(* CODESYS project fill.project

Project tree, tasks and I/O mapping:
  Device : 750-8111 PFC100, WAGO, order no. 750-8111, version 6.2.0.1
    application Application
      libraries: Standard, 3.5.18.0 (System)
      task DefaultTask (cyclic, interval T#10ms, priority 8) calls PLC_PRG
      Data types/
      Global Variables/
        global variables Variablen_Konfiguration
        global variables Globale_Variablen
      POUs/
        function block VALVE_VALID [CFC]
        function block BEMPTY [CFC]
        function block calc_progress [ST]
        function block calibrate [ST]
        function block ClearCommands [ST]
        function block conv_levelsensor [ST]
        function block copy_temperature [ST]
        function block EMPTY [CFC]
        function block FILL [CFC]
        function block FLUSH [CFC]
        function block WATERWARNING [CFC]
        program PLC_PRG [CFC]
        function block run_command [ST]
        function block SELECT_VALVE [ST]
        function block smooth [ST]
        function block TIMEOUT [ST]
        function block TIMEOUT_FB [CFC]
        Configuration/
          program MODBUS_CONFIGURATION [ST]
      Visualizations/
        visualisation temp
        visualisation PLC_VISU
      trace Sampling_Trace (task ): 
    Kbus : Kbus, WAGO, version 2.1.0.1
        unmapped channels: K-BUS diagnostics
      _750_497_16 : 750-497#16, WAGO, order no. 750-497, version 2.0.0.9
          unmapped channels: _PW 1, _PW 2, _PW 3, _PW 4, _PW 5, _PW 6, _PW 7, _PW 8
      _750_460_08 : 750-460#08, WAGO, order no. 750-460, version 2.0.0.9
          unmapped channels: _IINT 1, _IINT 2, _IINT 3, _IINT 4
      _750_430 : 750-430, WAGO, order no. 750-430, version 2.0.0.14
          unmapped channels: _IN
      _750_1504_1 : 750-1504, WAGO, order no. 750-1504, version 2.0.0.14
          unmapped channels: _OUT
      _750_1504 : 750-1504, WAGO, order no. 750-1504, version 2.0.0.14
          unmapped channels: _OUT
  GlobalImagePool
  text list GlobalTextList
*)

// Device/Application/Global Variables/Variablen_Konfiguration
VAR_CONFIG
END_VAR

// Device/Application/Global Variables/Globale_Variablen
VAR_GLOBAL

	(* 8x AI 0-10V *)
	ACTWEIGHT 		AT %IW0:INT; (* 0 Actual reservoir weight in digital units, evtl. with status byte *)
	RAINFILL1 		AT %IW1:INT; (* 1 Rainbucket filling in digital units, 2.2V / 0.305mV/DU is 100% *)
	RAINFILL2 		AT %IW2:INT; (* 2 Rainbucket filling in digital units, 2.2V / 0.305mV/DU is 100% *)
	AUX0				AT %IW3:INT;
	AUX1				AT %IW4:INT;
	AUX2				AT %IW5:INT;
	AUX3				AT %IW6:INT;
	AUX4				AT %IW7:INT;

	(*4x Pt100 *)
	PT100_1			AT %IW8:INT;
	PT100_2			AT %IW9:INT;
	PT100_3			AT %IW10:INT;
	PT100_4			AT %IW11:INT;

	(* 8x DI *)
	BTN_RESET_HW	AT %IX12.0:BOOL; (* 1 Stops the current action and cancels Warnings*)
	BTN_EMPTY_HW	AT %IX12.1:BOOL; (* 2 Empties the reservoir *)
	WATERWARN1	AT %IX12.4:BOOL; (* 5 Water sensor under mounting wall (not implemented) *)
	WATERWARN2	AT %IX12.5:BOOL; (* 6 Water sensor in fridge (not implemented) *)


	(* 8x DO *)
	P1_FWD 			AT %QX0.0:BOOL; (* Main pump forward *)
	P1_BCK 			AT %QX0.1:BOOL; (* Main pump backward *)
	VRin 				AT %QX0.2:BOOL; (* Flush / Fill selector valve VRin *)
	VRout 				AT %QX0.3:BOOL; (* 2/2 Valve at reservoir outlet, connected with pump 2 *)
	VRfridge 			AT %QX0.4:BOOL; (* 3/2 valve Fridge / Valve *)
	YSI600R_PWR	AT %QX0.5:BOOL; (* Relais to power YSI600R *)
	(*AUX_DO1  		AT %QX1.7:BOOL; *)

	(* 8x DO *)
	WWARN_LED		AT %QX1.0:BOOL;
	TIMEOUT_LED 	AT %QX1.1:BOOL; (* Indicates an unwanted timeout at empty or fill*)
	RUNNING_LED 	AT %QX1.2:BOOL; (* Indicates an unwanted timeout at empty or fill*)


	(* 8x DO - Input Valves, defined in SELECT_VALVE
		%QX1.0..7
	*)
	(* 8x DO - Input Valves, defined in SELECT_VALVE
		%QX1.8..15
	*)


	(* MERKER *)
	(* Commands *)
	BTN_RESET		AT %MX0.0:BOOL; (* Resets the current action *)
	BTN_FLUSH		AT %MX0.1:BOOL; (* Starts the fill sequence, when valve is selected*)
	BTN_FILL 			AT %MX0.2:BOOL; (* Starts the fill sequence when ACTWEIGHT<TGTWEIGHT*)
	BTN_EMPTY		AT %MX0.3:BOOL; (* Starts the empty sequence when ACTWEIGHT>TGTWEIGHT*)
       BTN_FRIDGE		AT %MX0.4:BOOL; (* Sets the fridge, use together with BTN_EMPTY*)
	BTN_BEMPTY		AT %MX0.5:BOOL; (* Runs backward empty (not implemented yet*)
	BTN_YSI600R		AT %MX0.6:BOOL; (* Switches the YSI600R on during flush*)
	BTN_CALIB		AT %MX0.7:BOOL; (* Calibrates the scale *)
	BTN_RAISE_TIMEOUT AT %MX0.8:BOOL; (* Indicates that a timeout should be raised *)
	(* Command arguments *)
	VALVE 				AT %MW1:INT; (*The actual valve number*)
	TGTWEIGHT 		AT %MW2:REAL;  (*target weight in ml *)
	TIMEOUT_VAL 	AT %MW4:TIME := t#10s; (* The timeout value *)

	(* Status *)
	ST_RUNNING		AT %MX6.0:BOOL;
	ST_TIMEOUT		AT %MX6.1:BOOL;
	ST_WWARN		AT %MX6.2:BOOL;
	ST_READY		AT %MX6.3:BOOL;
	ST_RESET		AT %MX6.4:BOOL;

	PROGRESS		AT %MW7:INT;
	AVGWEIGHT		AT %MW8:REAL := -1E10; (* Average weight in ml *)
	ELAPSED 			AT %MW10:TIME; (* The elapsed time *)
	RAINFILL1_out	AT %MW12:REAL;
	RAINFILL2_out	AT %MW14:REAL;
	(*Settings*)
	MAX_VALVE		AT %MW16:INT := 12; (* Maximum number of available valves *)
	WSMOOTH		AT %MW17:INT := 10; (* Smooth factor for low pass filter *)
	CALIB_OFFSET	AT %MW18:REAL := 0; (* Offset in digital units, when empty *)
	CALIB_GAIN		AT %MW20:REAL := 0.153; (* Gain of weight calibration in ml/DU *)

	(* Temperature *)
	TEMP1			     AT %MW22:INT;
	TEMP2			     AT %MW23:INT;
       TEMP3                  AT %MW24:INT;
       TEMP4                  AT %MW25:INT;

	START_WEIGHT: REAL;

END_VAR

// Device/Application/POUs/PLC_PRG
PROGRAM PLC_PRG
VAR

	VALVE_SELECTOR: SELECT_VALVE;
	WATERWARNING: WATERWARNING;
	weight_smooth: smooth;
	conv_rf1: conv_levelsensor;
	conv_rf2: conv_levelsensor;
	START_WEIGHT: REAL;
	CMD: run_command;
	_timeout: TIMEOUT;
	CP_TEMP: copy_temperature;
END_VAR
VAR // added by the converter: edge detectors and wires of the graphical bodies
    _w1 : ANY;
END_VAR

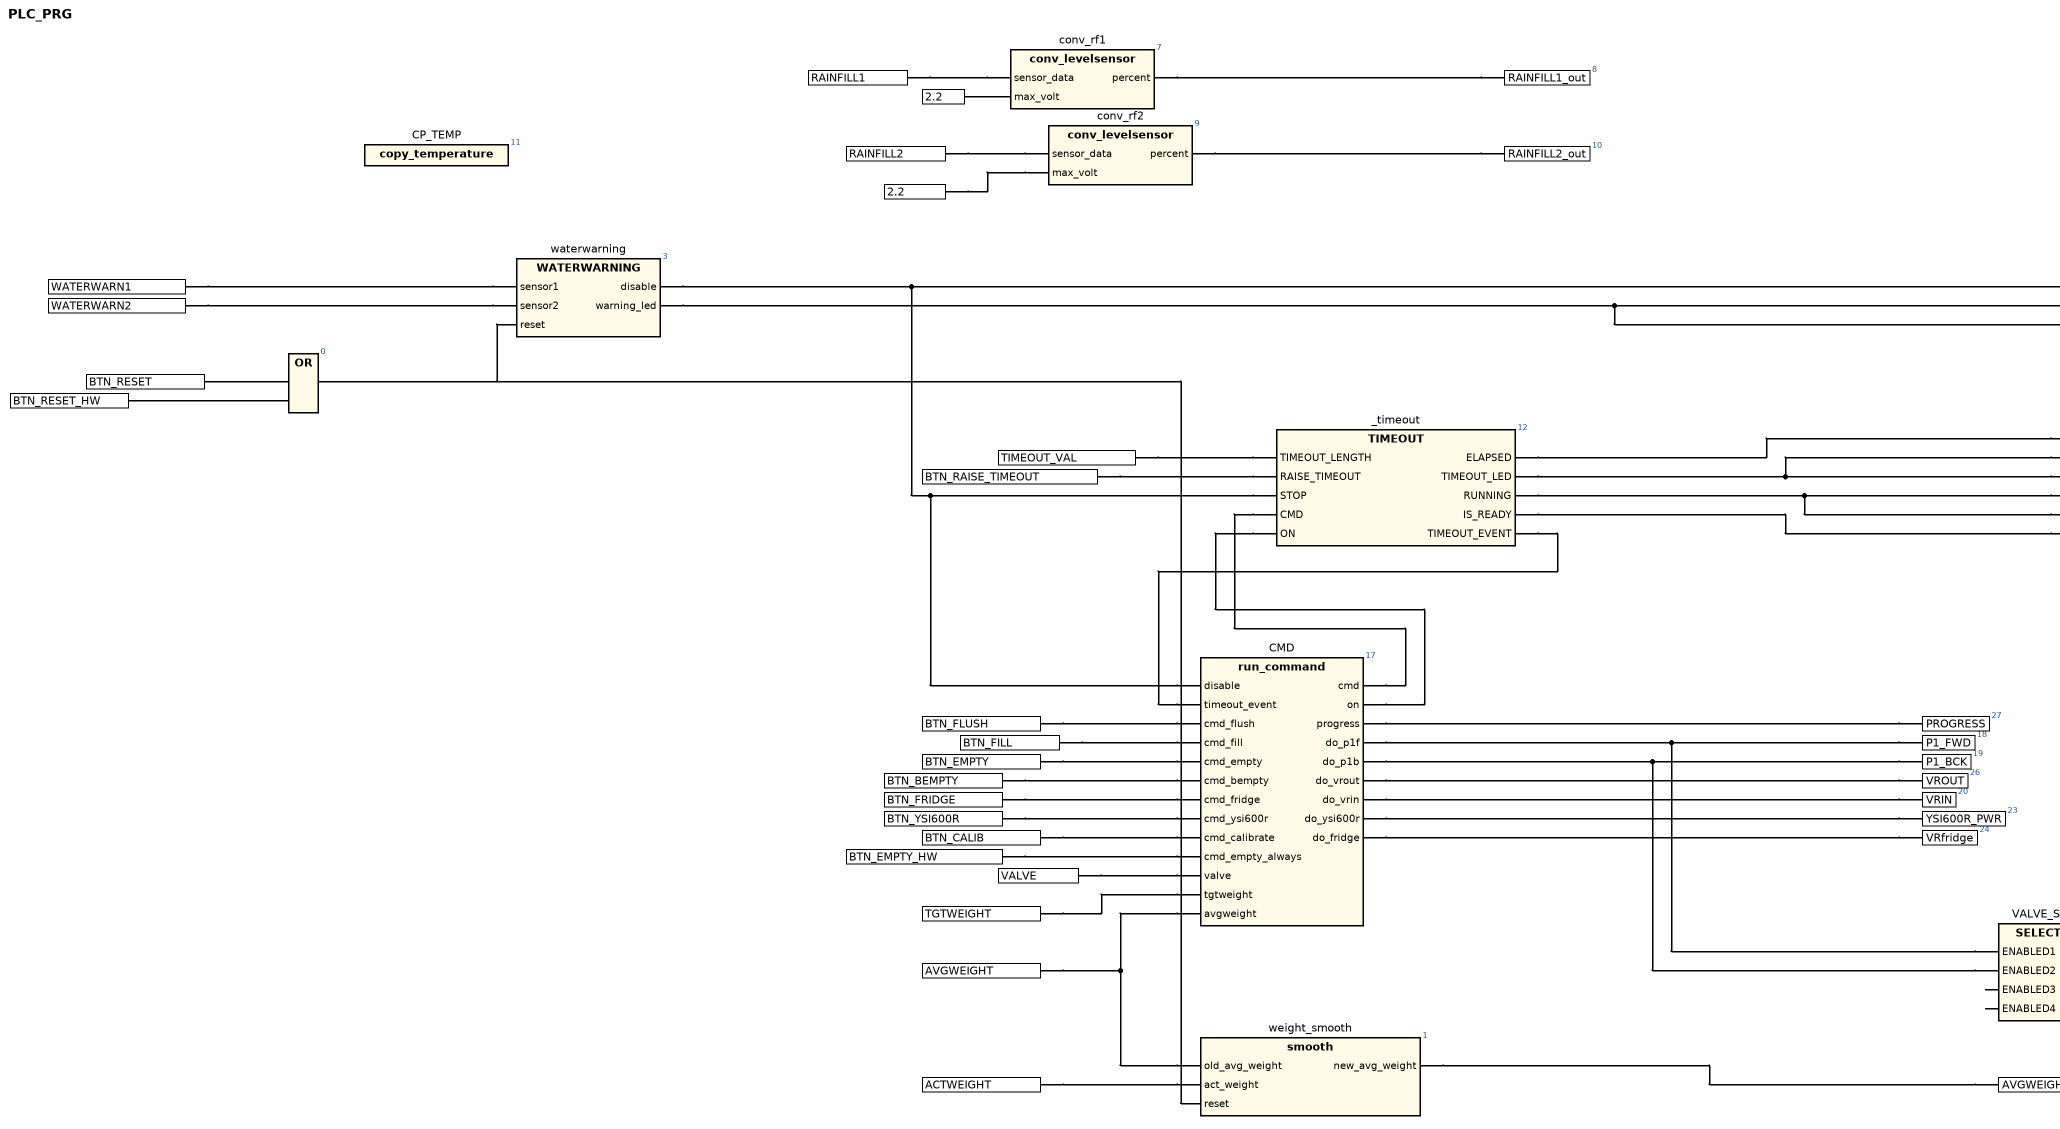
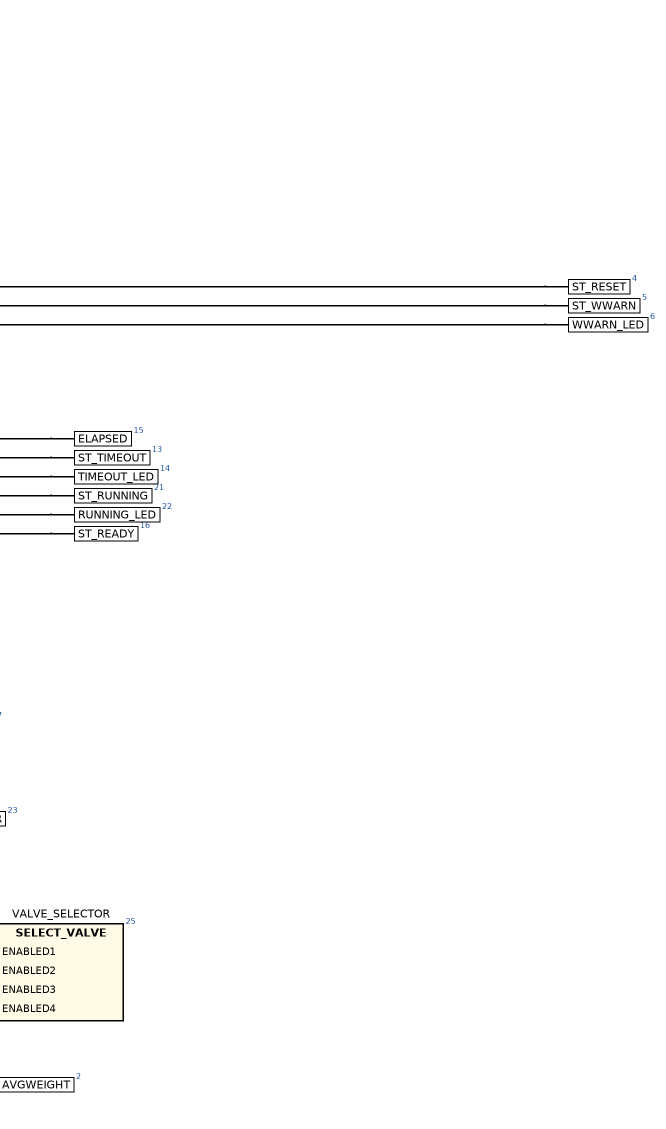
_w1 := BTN_RESET OR BTN_RESET_HW;
weight_smooth(old_avg_weight := AVGWEIGHT, act_weight := ACTWEIGHT, reset := _w1); // smooth
AVGWEIGHT := weight_smooth.new_avg_weight;
waterwarning(sensor1 := WATERWARN1, sensor2 := WATERWARN2, reset := _w1);
ST_RESET := waterwarning.disable;
ST_WWARN := waterwarning.warning_led;
WWARN_LED := waterwarning.warning_led;
conv_rf1(sensor_data := RAINFILL1, max_volt := 2.2); // conv_levelsensor
RAINFILL1_out := conv_rf1.percent;
conv_rf2(sensor_data := RAINFILL2, max_volt := 2.2); // conv_levelsensor
RAINFILL2_out := conv_rf2.percent;
CP_TEMP(); // copy_temperature
_timeout(
    TIMEOUT_LENGTH := TIMEOUT_VAL,
    RAISE_TIMEOUT := BTN_RAISE_TIMEOUT,
    STOP := waterwarning.disable,
    CMD := CMD.cmd,
    ON := CMD.on); // TIMEOUT
ST_TIMEOUT := _timeout.TIMEOUT_LED;
TIMEOUT_LED := _timeout.TIMEOUT_LED;
ELAPSED := _timeout.ELAPSED;
ST_READY := _timeout.IS_READY;
CMD(
    disable := waterwarning.disable,
    timeout_event := _timeout.TIMEOUT_EVENT,
    cmd_flush := BTN_FLUSH,
    cmd_fill := BTN_FILL,
    cmd_empty := BTN_EMPTY,
    cmd_bempty := BTN_BEMPTY,
    cmd_fridge := BTN_FRIDGE,
    cmd_ysi600r := BTN_YSI600R,
    cmd_calibrate := BTN_CALIB,
    cmd_empty_always := BTN_EMPTY_HW,
    valve := VALVE,
    tgtweight := TGTWEIGHT,
    avgweight := AVGWEIGHT); // run_command
P1_FWD := CMD.do_p1f;
P1_BCK := CMD.do_p1b;
VRIN := CMD.do_vrin;
ST_RUNNING := _timeout.RUNNING;
RUNNING_LED := _timeout.RUNNING;
YSI600R_PWR := CMD.do_ysi600r;
VRfridge := CMD.do_fridge;
VALVE_SELECTOR(ENABLED1 := CMD.do_p1f, ENABLED2 := CMD.do_p1b); // SELECT_VALVE
VROUT := CMD.do_vrout;
PROGRESS := CMD.progress;

END_PROGRAM

// Device/Application/POUs/smooth
FUNCTION_BLOCK smooth
VAR_INPUT
	old_avg_weight:REAL;
	act_weight:INT;
	reset:BOOL;
END_VAR
VAR_OUTPUT
	new_avg_weight:REAL;
END_VAR
VAR
	calib_w:REAL;
END_VAR


(* Calibrate actual weight *)

calib_w := act_weight  * CALIB_GAIN - CALIB_OFFSET;


IF old_avg_weight<-1E9 OR reset=TRUE THEN
	(* no data available, use actual value without lowpass*)
	new_avg_weight := calib_w;
ELSE
	(* Apply low pass filter if data is available *)
	new_avg_weight := old_avg_weight + (calib_w - old_avg_weight) / WSMOOTH;
END_IF

END_FUNCTION_BLOCK

// Device/Application/POUs/calibrate
FUNCTION_BLOCK calibrate
VAR_INPUT
END_VAR
VAR_OUTPUT
END_VAR
VAR
	Trigger:R_TRIG;
	avgw_du:REAL;
END_VAR

Trigger(CLK:=BTN_CALIB);
IF Trigger.Q THEN
	IF TGTWEIGHT>0 THEN
		(* uncalibrate smoothed avgweight *)
		avgw_du:=(AVGWEIGHT + CALIB_OFFSET)/CALIB_GAIN;
		(* calculate new gain *)
		CALIB_GAIN:= CALIB_GAIN * (CALIB_OFFSET + TGTWEIGHT)/(CALIB_OFFSET + AVGWEIGHT);
	ELSE
		CALIB_OFFSET := CALIB_OFFSET + AVGWEIGHT;
	END_IF
	BTN_CALIB:=FALSE;
END_IF

END_FUNCTION_BLOCK

// Device/Application/POUs/WATERWARNING
FUNCTION_BLOCK WATERWARNING
VAR_INPUT
	sensor1:BOOL;
	sensor2:BOOL;
	reset:BOOL;
END_VAR
VAR_OUTPUT
	disable:BOOL;
	warning_led:BOOL;
END_VAR
VAR
	sr_warning: SR;
	set_reset: SR;
END_VAR

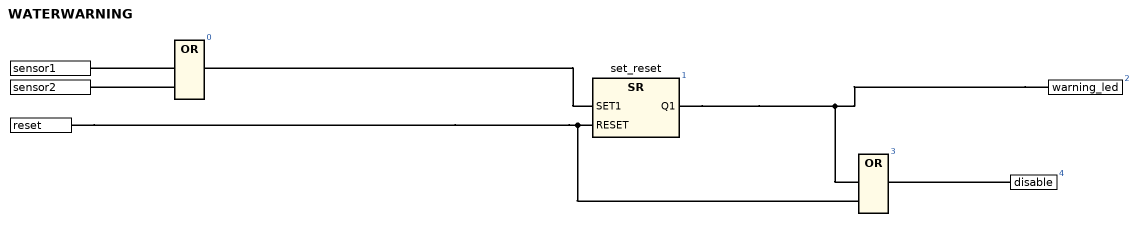
set_reset(SET1 := sensor1 OR sensor2, RESET := reset); // SR
warning_led := set_reset.Q1;
disable := set_reset.Q1 OR reset;

END_FUNCTION_BLOCK

// Device/Application/POUs/TIMEOUT
FUNCTION_BLOCK TIMEOUT
VAR_INPUT
	TIMEOUT_LENGTH:TIME;
	RAISE_TIMEOUT:BOOL; (* indicate timeout problem*)
	STOP:BOOL; (*reset button*)
	CMD:BOOL;
	ON:BOOL;
END_VAR
VAR_OUTPUT
	ELAPSED:TIME; (*Elapsed time*)
	TIMEOUT_LED:BOOL; (* Indicator LED for timeout events, only for fill and empty *)
	RUNNING:BOOL;
	IS_READY:BOOL;
	TIMEOUT_EVENT:BOOL; (* switches to TRUE when timeout is gone, feeds into reset of actions *)
END_VAR
VAR
	INDICATOR: RS;
	TIMEMACHINE: TON;
	RESET_IND: R_TRIG;
	latch_ready:RS;

END_VAR

(* Is a command running? *)
RUNNING := ON AND NOT STOP;

(* Get the time run, and output of timeevent and the elapsed time *)
TIMEMACHINE(IN:=RUNNING, PT:=TIMEOUT_LENGTH);
TIMEOUT_EVENT:=TIMEMACHINE.Q;
IF RUNNING THEN
	ELAPSED:=TIMEMACHINE.ET;
END_IF

(* check the timeout led *)
(* trigger on start *)
RESET_IND(CLK:=running);
INDICATOR(SET:=TIMEOUT_EVENT AND on AND RAISE_TIMEOUT,
			   RESET1:=RESET_IND.Q OR STOP OR NOT RAISE_TIMEOUT);

TIMEOUT_LED:=INDICATOR.Q1;

(* check is_ready *)
latch_ready(SET:=CMD, RESET1:=ON OR STOP OR NOT CMD);
IS_READY:=latch_ready.Q1;

END_FUNCTION_BLOCK

// Device/Application/POUs/FILL
FUNCTION_BLOCK FILL
VAR_INPUT
	START: BOOL; (* Triggers the start *)
	ACT_WEIGHT: REAL; (* Actual weight in DU *)
	TGT_WEIGHT: REAL; (* Target weight in DU *)
	RESET: BOOL;
	TIMEOUT_EVENT:BOOL;
	HAS_VALVE:BOOL;  (* Needs to be true for filling - true when a valve is set *)
	RUNNING:BOOL; (*TRUE when a task is running already*)
END_VAR
VAR_OUTPUT
	PUMP_FWD: BOOL;		(*Runs the pump forward to get water into the reservoir*)
	FILL_VR_In: BOOL;		(*Directs the inflow to the reservoir *)
END_VAR
VAR
	ENTPRELL_ZEIT: TIME :=t#1s;
	TON_ENTPRELL: TON;
	RS_FILL_ON: RS;
	trig: R_TRIG;
END_VAR
VAR // added by the converter: edge detectors and wires of the graphical bodies
    _w1, _w2 : BOOL;
    _w3 : REAL;
END_VAR

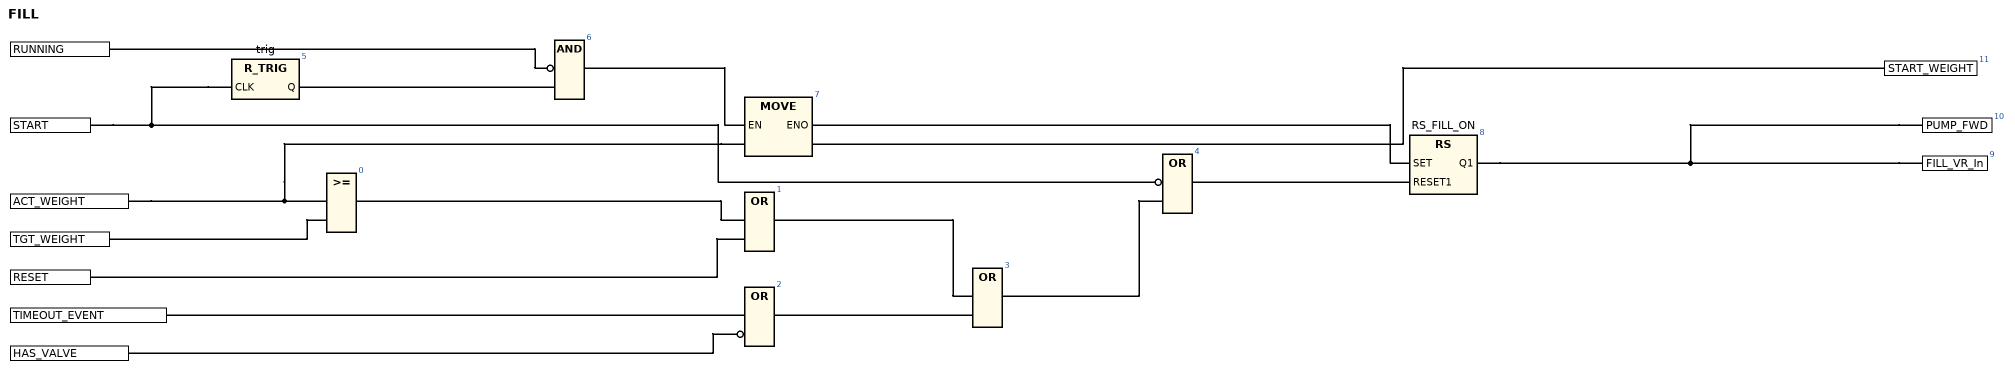
_w1 := NOT START OR ((ACT_WEIGHT >= TGT_WEIGHT OR RESET) OR (TIMEOUT_EVENT OR NOT HAS_VALVE));
trig(CLK := START); // R_TRIG
_w2 := NOT RUNNING AND trig.Q;
IF _w2 THEN _w3 := ACT_WEIGHT; END_IF
RS_FILL_ON(SET := _w2, RESET1 := _w1); // RS
FILL_VR_In := RS_FILL_ON.Q1;
PUMP_FWD := RS_FILL_ON.Q1;
START_WEIGHT := _w3;

END_FUNCTION_BLOCK

// Device/Application/POUs/EMPTY
FUNCTION_BLOCK EMPTY
VAR_INPUT
	START: BOOL;
	ACT_WEIGHT: REAL;
	TGT_WEIGHT: REAL;
	TO_FRIDGE: BOOL;
	RESET: BOOL;
	TIMEOUT_EVENT:BOOL;
	RUNNING:BOOL; (*TRUE when a task is running already*)

END_VAR
VAR_OUTPUT
	VROUT: BOOL;		(*Runs the pump forward to get water into the reservoir*)
	VFRIDGE: BOOL;
END_VAR
VAR
	ENTPRELL: TON;
	TON_ENTPRELL: TON;
	RS_FILL_ON: RS;
	RS_TO_FRIDGE: RS;
	trig: R_TRIG;
END_VAR
VAR // added by the converter: edge detectors and wires of the graphical bodies
    _w1, _w2, _w3 : BOOL;
    _w4 : REAL;
END_VAR

_w1 := (ACT_WEIGHT <= TGT_WEIGHT OR RESET) OR TIMEOUT_EVENT;
_w2 := NOT START OR _w1;
trig(CLK := START); // R_TRIG
_w3 := NOT RUNNING AND trig.Q;
IF _w3 THEN _w4 := ACT_WEIGHT; END_IF
START_WEIGHT := _w4;
RS_FILL_ON(SET := _w3, RESET1 := _w2); // RS
VROUT := RS_FILL_ON.Q1;
RS_TO_FRIDGE(SET := TO_FRIDGE, RESET1 := _w1); // RS
VFRIDGE := RS_FILL_ON.Q1 AND RS_TO_FRIDGE.Q1;

END_FUNCTION_BLOCK

// Device/Application/POUs/run_command
FUNCTION_BLOCK run_command
VAR_INPUT
	disable:BOOL;
	timeout_event:BOOL;
	cmd_flush:BOOL;
	cmd_fill:BOOL;
	cmd_empty:BOOL;
	cmd_bempty:BOOL;
	cmd_fridge:BOOL;
	cmd_ysi600r: BOOL;
	cmd_calibrate:BOOL;
	cmd_empty_always:BOOL;
	valve:INT;
	tgtweight:REAL;
	avgweight:REAL;

END_VAR
VAR_OUTPUT
	cmd: BOOL;
	on:BOOL;
	progress:INT;
	do_p1f:BOOL;
	do_p1b:BOOL;
	do_vrout:BOOL;
	do_vrin:BOOL;
	do_ysi600r:BOOL;
	do_fridge: BOOL;
END_VAR
VAR
	_is_running:BOOL;
	_flush: FLUSH;
	_fill: FILL;
      _empty: EMPTY;
      _bempty: BEMPTY;
      _valve_valid: VALVE_VALID;
	_clear_commands: ClearCommands;
	_calibrate_trigger: R_TRIG;
END_VAR

_calibrate_trigger(CLK:=cmd_calibrate);
_is_running:=P1_BCK OR P1_FWD OR VRout;
_clear_commands(disable:=disable);

IF  disable THEN
	do_p1f:=FALSE;
	do_p1b:=FALSE;
	do_fridge:=FALSE;
	do_ysi600r:=FALSE;
	do_vrout:=FALSE;
	do_vrin:=FALSE;
END_IF

IF _calibrate_trigger.Q AND NOT _is_running THEN
	IF tgtweight>0 THEN
		(* calculate new gain *)
		CALIB_GAIN:= CALIB_GAIN * (CALIB_OFFSET + TGTWEIGHT)/(CALIB_OFFSET + AVGWEIGHT);
	ELSE
		CALIB_OFFSET := CALIB_OFFSET + AVGWEIGHT + 2.0;
	END_IF

	BTN_CALIB:=FALSE;

END_IF

_valve_valid(valve_id:=valve);
_flush(START:=cmd_flush,
             HAS_VALVE:=_valve_valid.is_valid,
		RESET:=disable,
		TIMEOUT_EVENT:=timeout_event,
		RUNNING:=_is_running,
		YSI600R_ENABLE:=cmd_ysi600r);

_fill(START:=cmd_fill,
             HAS_VALVE:=_valve_valid.is_valid,
		RESET:=disable,
		TIMEOUT_EVENT:=timeout_event,
		RUNNING:=_is_running,
		ACT_WEIGHT:=avgweight,
		TGT_WEIGHT:=tgtweight);

_bempty(START:=cmd_bempty,
             HAS_VALVE:=_valve_valid.is_valid,
		RESET:=disable,
		TIMEOUT_EVENT:=timeout_event,
		RUNNING:=_is_running,
		ACT_WEIGHT:=avgweight,
		TGT_WEIGHT:=tgtweight);

_empty(START:=cmd_empty,
             TO_FRIDGE:=cmd_fridge,
		RESET:=disable,
		TIMEOUT_EVENT:=timeout_event,
		RUNNING:=_is_running,
		ACT_WEIGHT:=avgweight,
		TGT_WEIGHT:=tgtweight);

do_p1f:=_flush.PUMP_FWD OR _fill.PUMP_FWD;
do_p1b:=_bempty.PUMP_BACK;
do_vrout:=_empty.VROUT OR cmd_empty_always;
do_vrin:=_fill.FILL_VR_In OR _bempty.FILL_VR_In;
do_ysi600r:=_flush.YSI600R;
do_fridge:=_empty.VFRIDGE;

on:=do_p1f OR do_p1b OR do_vrout;
cmd:=cmd_flush OR cmd_fill OR cmd_empty OR cmd_bempty;

IF cmd_flush AND elapsed>T#0ms THEN
	(* Flush progress by time, when running has stopped, elapsed is zero but progress should stay at 10000 c% *)
	progress:=LIMIT(0, DWORD_TO_INT((10000 * TIME_TO_DWORD(ELAPSED) / TIME_TO_DWORD(TIMEOUT_VAL))), 10000);

ELSIF (cmd_fill OR cmd_empty OR cmd_bempty) AND _is_running THEN
	progress:=LIMIT(0, 10000 - REAL_TO_INT((10000 * (avgweight-tgtweight)/(START_WEIGHT-tgtweight))), 10000);
END_IF

END_FUNCTION_BLOCK

// Device/Application/POUs/FLUSH

FUNCTION_BLOCK FLUSH
VAR_INPUT
	START: BOOL;
	HAS_VALVE:BOOL;
	RESET: BOOL;
	TIMEOUT_EVENT:BOOL;
	YSI600R_ENABLE: BOOL;
	RUNNING:BOOL;
END_VAR
VAR_OUTPUT
	PUMP_FWD: BOOL;		(*Runs the pump forward to get water into the reservoir*)
	YSI600R: BOOL;
END_VAR
VAR
	RS_FLUSH_ON: RS;
	RS_YSI_ENABLE: RS;
	trig: R_TRIG;
END_VAR
VAR // added by the converter: edge detectors and wires of the graphical bodies
    _w1, _w2, _w3 : BOOL;
END_VAR

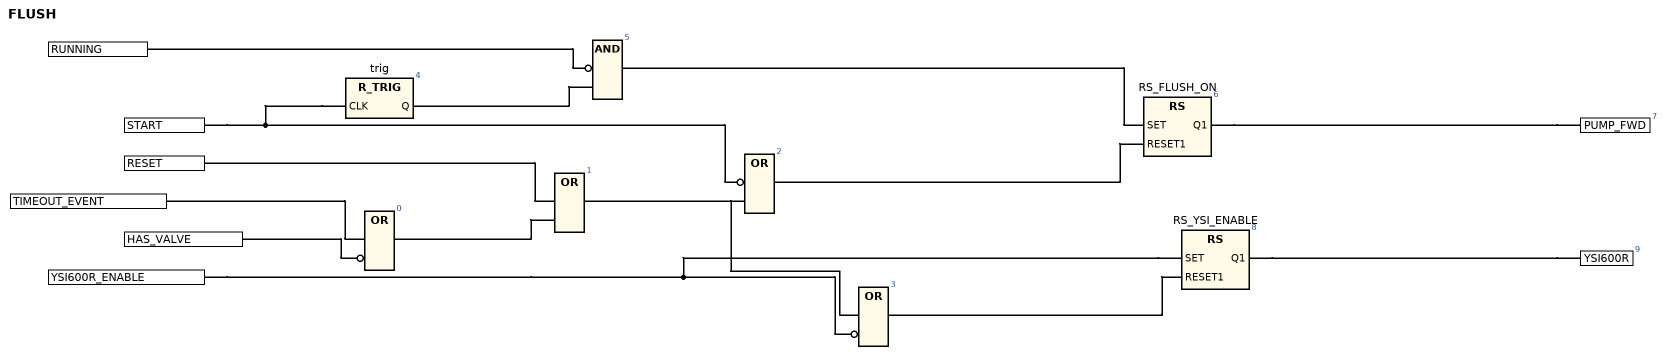
_w1 := RESET OR (TIMEOUT_EVENT OR NOT HAS_VALVE);
_w2 := NOT START OR _w1;
_w3 := _w1 OR NOT YSI600R_ENABLE;
trig(CLK := START); // R_TRIG
RS_FLUSH_ON(SET := NOT RUNNING AND trig.Q, RESET1 := _w2); // RS
PUMP_FWD := RS_FLUSH_ON.Q1;
RS_YSI_ENABLE(SET := YSI600R_ENABLE, RESET1 := _w3); // RS
YSI600R := RS_YSI_ENABLE.Q1;

END_FUNCTION_BLOCK

// Device/Application/POUs/BEMPTY
FUNCTION_BLOCK BEMPTY
VAR_INPUT
	START: BOOL; (* Triggers the start *)
	ACT_WEIGHT: REAL; (* Actual weight in DU *)
	TGT_WEIGHT: REAL; (* Target weight in DU *)
	RESET: BOOL;
	TIMEOUT_EVENT:BOOL;
	HAS_VALVE:BOOL;  (* Needs to be true for filling - true when a valve is set *)
	RUNNING:BOOL; (*TRUE when a task is running already*)
END_VAR
VAR_OUTPUT
	PUMP_BACK: BOOL;
	FILL_VR_In: BOOL;		(*Directs the inflow to the reservoir *)
END_VAR
VAR
	ENTPRELL_ZEIT: TIME :=t#1s;
	TON_ENTPRELL: TON;
	RS_FILL_ON: RS;
	trig: R_TRIG;
END_VAR
VAR // added by the converter: edge detectors and wires of the graphical bodies
    _w1, _w2 : BOOL;
    _w3 : REAL;
END_VAR

_w1 := NOT START OR ((ACT_WEIGHT <= TGT_WEIGHT OR RESET) OR (TIMEOUT_EVENT OR NOT HAS_VALVE));
trig(CLK := START); // R_TRIG
_w2 := NOT RUNNING AND trig.Q;
IF _w2 THEN _w3 := ACT_WEIGHT; END_IF
START_WEIGHT := _w3;
RS_FILL_ON(SET := _w2, RESET1 := _w1); // RS
FILL_VR_In := RS_FILL_ON.Q1;
PUMP_BACK := RS_FILL_ON.Q1;

END_FUNCTION_BLOCK

// Device/Application/POUs/VALVE_VALID
FUNCTION_BLOCK VALVE_VALID
VAR_INPUT
	valve_id:INT;
END_VAR
VAR_OUTPUT
	is_valid:BOOL;
END_VAR
VAR
END_VAR
VAR CONSTANT
	zero:WORD := 0;
END_VAR

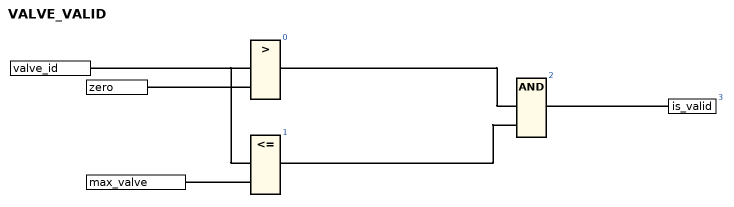
is_valid := valve_id > zero AND valve_id <= max_valve;

END_FUNCTION_BLOCK

// Device/Application/POUs/ClearCommands
FUNCTION_BLOCK ClearCommands
VAR_INPUT
	disable: BOOL;
END_VAR
VAR_OUTPUT
END_VAR
VAR
END_VAR


IF (disable) THEN
	BTN_RESET := FALSE;
	BTN_FLUSH := FALSE;
	BTN_FILL := FALSE;
	BTN_EMPTY := FALSE;
       BTN_FRIDGE := FALSE;
	BTN_BEMPTY := FALSE;
	BTN_YSI600R := FALSE;
	BTN_CALIB := FALSE;
	ST_READY := FALSE;

END_IF

END_FUNCTION_BLOCK

// Device/Application/POUs/SELECT_VALVE
FUNCTION_BLOCK SELECT_VALVE
VAR_INPUT

	ENABLED1:BOOL:=FALSE;
	ENABLED2:BOOL:=FALSE;
	ENABLED3:BOOL := FALSE;
	ENABLED4:BOOL := FALSE;
END_VAR

VAR_OUTPUT
END_VAR
VAR
END_VAR


IF (ENABLED1 OR ENABLED2 OR ENABLED3 OR ENABLED4) THEN
	CASE VALVE OF
		1: %QX2.0 := TRUE;
		2: %QX2.1 := TRUE;
		3: %QX2.2 := TRUE;
		4: %QX2.3 := TRUE;
		5: %QX2.4 := TRUE;
		6: %QX2.5 := TRUE;
		7: %QX2.6 := TRUE;
		8: %QX2.7 := TRUE;
		9: %QX3.0 := TRUE;
		10: %QX3.1 := TRUE;
		11: %QX3.2 := TRUE;
		12: %QX3.3 := TRUE;
		13: %QX3.4 := TRUE;
		14: %QX3.5 := TRUE;
		15: %QX3.6 := TRUE;
		16: %QX3.7 := TRUE;
	END_CASE
ELSE
	%QX2.0 := FALSE;
	%QX2.1 := FALSE;
	%QX2.2 := FALSE;
	%QX2.3 := FALSE;
	%QX2.4 := FALSE;
	%QX2.5 := FALSE;
	%QX2.6 := FALSE;
	%QX2.7 := FALSE;
	%QX3.0 := FALSE;
	%QX3.1 := FALSE;
	%QX3.2 := FALSE;
	%QX3.3 := FALSE;
	%QX3.4 := FALSE;
	%QX3.5 := FALSE;
	%QX3.6 := FALSE;
	%QX3.7 := FALSE;
END_IF

END_FUNCTION_BLOCK

// Device/Application/POUs/conv_levelsensor
FUNCTION_BLOCK conv_levelsensor
(* converts level sensor raw data to % of max. voltage *)
VAR_INPUT
	sensor_data:INT; (* The raw data from the sensor in digital units*)
	max_volt:REAL:=10.0; (* The max voltage of the sensor *)
END_VAR
VAR_OUTPUT
	percent:REAL; (* the percentage of the gain *)
END_VAR
VAR

	volt: REAL;
END_VAR

volt := 10 * sensor_data / 32767.0;
percent := volt / max_volt * 100.0;

END_FUNCTION_BLOCK

// Device/Application/POUs/copy_temperature
FUNCTION_BLOCK copy_temperature
VAR_INPUT
END_VAR
VAR_OUTPUT
END_VAR
VAR
END_VAR


TEMP1:=PT100_1;
TEMP2:=PT100_2;
TEMP3:=PT100_3;
TEMP4:=PT100_4;

(* do conversion of rainfill here *)

END_FUNCTION_BLOCK

// Device/Application/POUs/calc_progress
FUNCTION_BLOCK calc_progress
VAR_INPUT
END_VAR
VAR_OUTPUT
	progress:WORD;
END_VAR
VAR
END_VAR


IF BTN_FLUSH=TRUE AND ELAPSED>T#0ms THEN
	(* Flush progress by time, when running has stopped, elapsed is zero but progress should stay at 10000 c% *)
	progress:=LIMIT(0, DWORD_TO_INT((10000 * TIME_TO_DWORD(ELAPSED) / TIME_TO_DWORD(TIMEOUT_VAL))), 10000);

ELSIF (BTN_FILL=TRUE OR BTN_EMPTY=TRUE OR BTN_BEMPTY=TRUE)	AND ST_RUNNING=TRUE THEN
	progress:=LIMIT(0, 10000 - REAL_TO_INT((10000 * (AVGWEIGHT-TGTWEIGHT)/(START_WEIGHT-TGTWEIGHT))), 10000);


END_IF

END_FUNCTION_BLOCK

// Device/Application/POUs/TIMEOUT_FB
FUNCTION_BLOCK TIMEOUT_FB
VAR_INPUT
	TIMEOUT_LENGTH:TIME;
	FLUSH:BOOL; (* Driven by flush pump signal*)
	FILL:BOOL; (* Driven by fill pump signal*)
	EMPTY:BOOL; (*Driven by VRout signal*)
	BEMPTY:BOOL; (* Driven by P1_BCK *)
	STOP:BOOL; (*reset button*)
END_VAR
VAR_OUTPUT
	ELAPSED:TIME; (*Elapsed time*)
	TIMEOUT_EVENT:BOOL; (* switches to TRUE when timeout is gone, feeds into reset of actions *)
	TIMEOUT_LED:BOOL; (* Indicator LED for timeout events, only for fill and empty *)
	RUNNING:BOOL;
END_VAR
VAR
	INDICATOR: RS;
	TIMEMACHINE: TON;
	RESET_IND: R_TRIG;
END_VAR
VAR // added by the converter: edge detectors and wires of the graphical bodies
    _w1, _w2, _w3, _w5 : BOOL;
    _w4 : ANY;
END_VAR

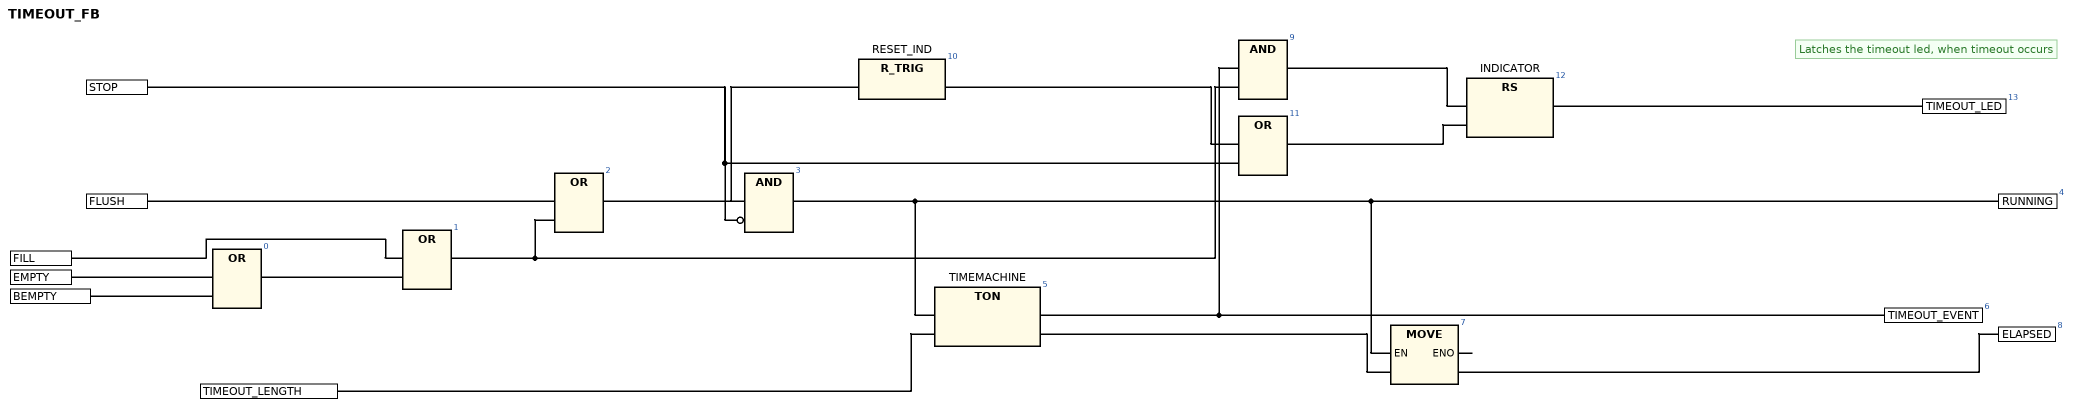
_w1 := FILL OR (EMPTY OR BEMPTY);
_w2 := FLUSH OR _w1;
_w3 := _w2 AND NOT STOP;
RUNNING := _w3;
TIMEMACHINE(_in1 := _w3, _in2 := TIMEOUT_LENGTH); // TON
TIMEOUT_EVENT := TIMEMACHINE._out1;
IF _w3 THEN _w4 := TIMEMACHINE._out2; END_IF
ELAPSED := _w4;
_w5 := TIMEMACHINE._out1 AND _w1;
RESET_IND(_in1 := _w2); // R_TRIG
INDICATOR(_in1 := _w5, _in2 := RESET_IND._out1 OR STOP); // RS
// Latches the timeout led, when timeout occurs
TIMEOUT_LED := INDICATOR._out1;

END_FUNCTION_BLOCK

// Device/Application/POUs/Configuration/MODBUS_CONFIGURATION
PROGRAM MODBUS_CONFIGURATION        
VAR                                
END_VAR

(*                                 
   <?xml version="1.0" encoding="UTF-16" standalone="yes"?>
<network xml_structure_version="1" xml_feature_version="1">
	<generator_settings minRTUTaskCycleTimeMs="5" minEthaskCycleTimeMs="5" ethSlaveMultiplier="0.1" rtuInterfaceMultiplier="0.1" taskGeneration="false"/>
</network>
                              
*)                                 
;

END_PROGRAM

// Device/Application/Visualizations/temp
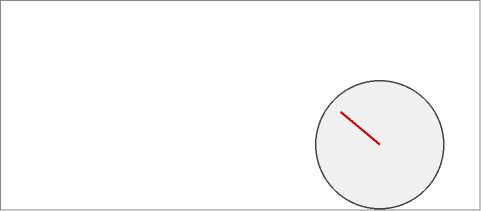
VISUALIZATION temp  // 481x211
    Meter (280,80 199x129), scale format: %.1f, scale 0..500
        p518627256: degC
END_VISUALIZATION

// Device/Application/Visualizations/PLC_VISU
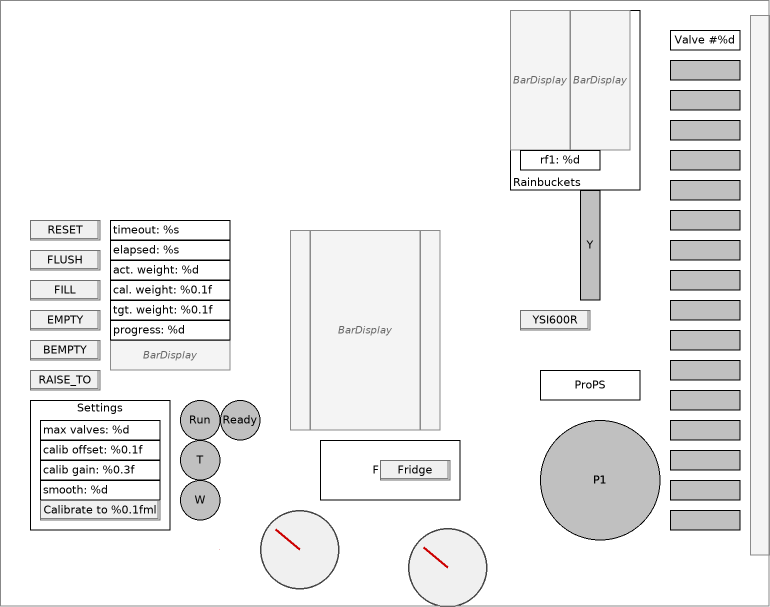
VISUALIZATION PLC_VISU  // 770x607
    Rectangle (510,10 130x180), "Rainbuckets"
    Rectangle (30,400 140x130), "Settings"
    RoundedRectangle (670,60 70x20), colour toggle: %QX1.0
    RoundedRectangle (670,90 70x20), colour toggle: %QX1.1
    RoundedRectangle (670,120 70x20), colour toggle: %QX1.2
    RoundedRectangle (670,150 70x20), colour toggle: %QX1.3
    RoundedRectangle (670,180 70x20), colour toggle: %QX1.4
    RoundedRectangle (670,210 70x20), colour toggle: %QX1.5
    RoundedRectangle (670,240 70x20), colour toggle: %QX1.6
    RoundedRectangle (670,270 70x20), colour toggle: %QX1.7
    RoundedRectangle (670,300 70x20), colour toggle: %QX1.8
    RoundedRectangle (670,330 70x20), colour toggle: %QX1.9
    RoundedRectangle (670,360 70x20), colour toggle: %QX1.10
    RoundedRectangle (670,390 70x20), colour toggle: %QX1.11
    RoundedRectangle (670,420 70x20), colour toggle: %QX1.12
    RoundedRectangle (670,450 70x20), colour toggle: %QX1.13
    RoundedRectangle (670,480 70x20), colour toggle: %QX1.14
    RoundedRectangle (670,510 70x20), colour toggle: %QX1.15
    Button (30,220 70x20), "RESET"
        tap Globale_Variablen.BTN_RESET
    BarDisplay (310,230 110x200), value: AVGWEIGHT, scale format: %.0f, scale 0..1000
        p518627256: ml
    Scrollbar (420,230 20x200)
        p1057716461: Globale_Variablen.TGTWEIGHT
    Button (30,250 70x20), "FLUSH", pressed state: Globale_Variablen.BTN_FLUSH
        toggle Globale_Variablen.BTN_FLUSH
    Button (30,280 70x20), "FILL", pressed state: Globale_Variablen.BTN_FILL
        toggle Globale_Variablen.BTN_FILL
    Polyline (540,480), colour toggle: Globale_Variablen.VRin
    Button (30,310 70x20), "EMPTY", pressed state: Globale_Variablen.BTN_EMPTY
        toggle Globale_Variablen.BTN_EMPTY
    Scrollbar (750,15 20x540)
        p1057716461: Globale_Variablen.VALVE
    Ellipse (180,400 40x40), "Run", colour toggle: Globale_Variablen.RUNNING_LED
    Ellipse (180,440 40x40), "T", colour toggle: Globale_Variablen.TIMEOUT_LED
    Ellipse (180,480 40x40), "W", colour toggle: Globale_Variablen.WWARN_LED
    Polygon (590,260), colour toggle: Globale_Variablen.VRin
    Rectangle (320,440 140x60), "Fridge", colour toggle: Globale_Variablen.VRfridge
    Polyline (360,490), colour toggle: Globale_Variablen.VRout
    Button (380,460 70x20), "Fridge", pressed state: Globale_Variablen.BTN_FRIDGE
        toggle Globale_Variablen.BTN_FRIDGE
    Button (520,310 70x20), "YSI600R", pressed state: Globale_Variablen.BTN_YSI600R
        toggle Globale_Variablen.BTN_YSI600R
    RoundedRectangle (580,190 20x110), "Y", colour toggle: Globale_Variablen.YSI600R_PWR
    Rectangle (110,240 120x20), "elapsed: %s", text variable: Globale_Variablen.ELAPSED
    Rectangle (110,220 120x20), "timeout: %s", text variable: Globale_Variablen.TIMEOUT_VAL
        OnMouseDown: write the text variable via Edit
    Ellipse (540,420 120x120), "P1", colour toggle: Globale_Variablen.P1_FWD
    RoundedRectangle (670,30 70x20), "Valve #%d", text variable: Globale_Variablen.VALVE
        OnMouseDown: write the text variable via Edit
    BarDisplay (510,10 60x140), value: RAINFILL1_out, scale format: %.0f, scale 0..100
        p518627256: %
    Rectangle (110,260 120x20), "act. weight: %d", text variable: Globale_Variablen.ACTWEIGHT
    Rectangle (110,300 120x20), "tgt. weight: %0.1f", text variable: Globale_Variablen.TGTWEIGHT
        OnMouseDown: write the text variable via Edit
    RoundedRectangle (540,370 100x30), "ProPS"
    Scrollbar (290,230 20x200)
        p1057716461: Globale_Variablen.ACTWEIGHT
    Rectangle (40,420 120x20), "max valves: %d", text variable: Globale_Variablen.MAX_VALVE
        OnMouseDown: write the text variable via Edit, min 1, max 16
    Rectangle (40,440 120x20), "calib offset: %0.1f", text variable: Globale_Variablen.CALIB_OFFSET
        OnMouseDown: write the text variable via Edit
    Rectangle (40,460 120x20), "calib gain: %0.3f", text variable: Globale_Variablen.CALIB_GAIN
        OnMouseDown: write the text variable via Edit
    Rectangle (40,480 120x20), "smooth: %d", text variable: Globale_Variablen.WSMOOTH
        OnMouseDown: write the text variable via Edit
    Button (40,500 120x20), "Calibrate to %0.1fml", text variable: Globale_Variablen.TGTWEIGHT
        tap Globale_Variablen.BTN_CALIB
    Rectangle (110,280 120x20), "cal. weight: %0.1f", text variable: Globale_Variablen.AVGWEIGHT
    Button (30,340 70x20), "BEMPTY", pressed state: Globale_Variablen.BTN_BEMPTY
        toggle Globale_Variablen.BTN_BEMPTY
    Ellipse (540,420 120x120), "P1", colour toggle: Globale_Variablen.P1_BCK
    BarDisplay (110,340 120x30), value: PROGRESS, scale format: %.0f, scale 0..10000
    Rectangle (110,320 120x20), "progress: %d", text variable: Globale_Variablen.TIMEOUT_VAL
        OnMouseDown: write the text variable via Edit
    BarDisplay (570,10 60x140), value: RAINFILL2_out, scale format: %.0f, scale 0..100
        p518627256: %
    Rectangle (520,150 80x20), "rf1: %d", text variable: Globale_Variablen.RAINFILL1
    Button (30,370 70x20), "RAISE_TO", pressed state: Globale_Variablen.BTN_RAISE_TIMEOUT
        toggle Globale_Variablen.BTN_RAISE_TIMEOUT
    Ellipse (220,400 40x40), "Ready", colour toggle: Globale_Variablen.ST_READY
    Meter (220,550 -1x-1), value: TEMP1, scale format: %.1f, scale 0..60
        p518627256: °C
    Meter (230,510 139x79), value: TEMP1, scale format: %.0f, scale 0..500
        p518627256: °C
    Meter (378,528 139x79), value: TEMP3, scale format: %.0f, scale 0..500
        p518627256: °C
END_VISUALIZATION
